Staubli VAL3: yes_no.pgx

public program yes_no(string x_sMessage, string& x_sYesNo[], bool& x_bResult[])
  local num i
  local string l_sButton[2]
begin
  //
  // write a yes no question dialog
  //
  if x_sYesNo!=""
    l_sButton[0]=x_sYesNo
  else
    l_sButton[0]="Yes"
  endIf
  //
  if x_sYesNo[1]!=""
    l_sButton[1]=x_sYesNo[1]
  else
    l_sButton[1]="No"
  endIf
  // question Dialog
  call questionDialog(x_sMessage,l_sButton,i)
  // press F8->YES or ENTER
  if i==1 or i==0
    x_bResult=true
  else
    // press escape or F7->NO
    x_bResult=false
  endIf
end
